// TIA Portal V17 export
// export: Created 2024-08-29T18:23:50.969703Z, ExportSetting WithDefaults, DisplayName Totally Integrated Automation Portal, DisplayVersion V17 Update 7, DisplayName TIA Portal Openness, DisplayVersion V17 Update 7, DisplayName TIA Portal Version Control Interface, DisplayVersion V17, DisplayName SINAMICS Startdrive Advanced, DisplayVersion V17 SP2, DisplayName SINAMICS Startdrive G110M, G120, G120C, G120D, G120P, G115D, DisplayVersion V17 SP2, DisplayName SINAMICS Startdrive G130, G150, S120, S150, SINAMICS MV, S210, DisplayVersion V17 SP2, DisplayName STEP 7 Professional, DisplayVersion V17 Update 7, DisplayName STEP 7 Safety, DisplayVersion V17 Update 6, DisplayName WinCC Advanced / Unified PC, DisplayVersion V17 Update 7
VAR_GLOBAL   // PLC tag table "printerMemory"
   reqPrint AT %M4000.0 : Bool;
   reqLastLabel AT %M4000.1 : Bool;
   resetPrinterErrors AT %M4000.2 : Bool;
   printBlackLabel AT %M4000.3 : Bool;
   resetPrinterCounter AT %M4000.4 : Bool;
   hmiSavePrinterReference AT %M4000.5 : Bool;
   hmiReadPrinterReference AT %M4000.6 : Bool;
END_VAR
